// SIMATIC STEP 7 (V5.x) project PID_INS
// program: S7 Program(1)

SYMBOL_TABLE
"PID_L"	FB 136	FB 136	// Регулирования уровня в резервуаре активного ила
END_SYMBOL_TABLE

FUNCTION_BLOCK "PID_L"	// FB 136
AUTHOR : ETSystem
VERSION : 0.1
VAR_INPUT
  MAN_ON : BOOL ;
  P_SEL : BOOL ;
  I_SEL : BOOL ;
  D_SEL : BOOL ;
  SP_INT : REAL ;
  PV_IN : REAL ;
  MAN : REAL ;
  K_GAIN : REAL ;
  TI : TIME ;
  TD : TIME ;
  DEAD_BANDW : REAL ;
  LMN_HLM : REAL ;
  LMN_LLM : REAL ;
END_VAR
VAR_OUTPUT
  LMN : REAL ;
  PV : REAL ;
  ER : REAL ;
END_VAR
BEGIN
NETWORK
TITLE =
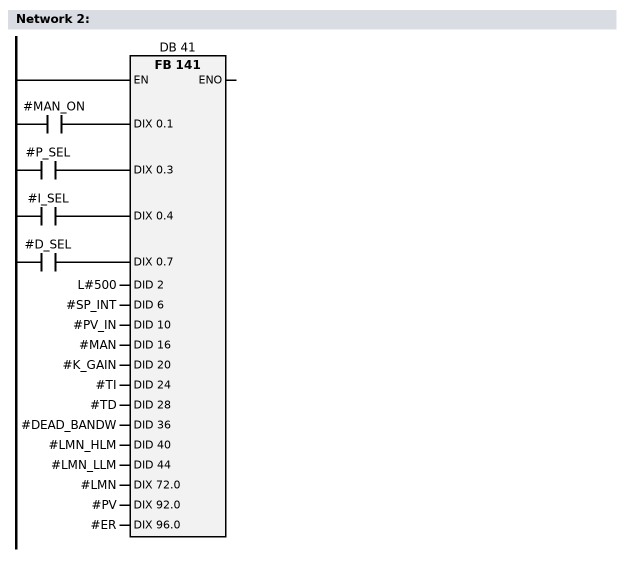
NETWORK
TITLE =
      A     #MAN_ON;
      =     L 0.1;
      BLD   103;
      A     #P_SEL;
      =     L 0.3;
      BLD   103;
      A     #I_SEL;
      =     L 0.4;
      BLD   103;
      A     #D_SEL;
      =     L 0.7;
      BLD   103;
      CALL  FB 141 , DB 41 (
           DIX 0.1                  := L 0.1,
           DIX 0.3                  := L 0.3,
           DIX 0.4                  := L 0.4,
           DIX 0.7                  := L 0.7,
           DID 2                    := L#500,
           DID 6                    := #SP_INT,
           DID 10                   := #PV_IN,
           DID 16                   := #MAN,
           DID 20                   := #K_GAIN,
           DID 24                   := #TI,
           DID 28                   := #TD,
           DID 36                   := #DEAD_BANDW,
           DID 40                   := #LMN_HLM,
           DID 44                   := #LMN_LLM,
           DIX 72.0                 := #LMN,
           DIX 92.0                 := #PV,
           DIX 96.0                 := #ER);
      NOP   0;
END_FUNCTION_BLOCK

ORGANIZATION_BLOCK OB 1
TITLE = "Main Program Sweep (Cycle)"
VERSION : 0.1
VAR_TEMP
  OB1_EV_CLASS : BYTE ;	//Bits 0-3 = 1 (Coming event), Bits 4-7 = 1 (Event class 1)
  OB1_SCAN_1 : BYTE ;	//1 (Cold restart scan 1 of OB 1), 3 (Scan 2-n of OB 1)
  OB1_PRIORITY : BYTE ;	//Priority of OB Execution
  OB1_OB_NUMBR : BYTE ;	//1 (Organization block 1, OB1)
  OB1_RESERVED_1 : BYTE ;	//Reserved for system
  OB1_RESERVED_2 : BYTE ;	//Reserved for system
  OB1_PREV_CYCLE : INT ;	//Cycle time of previous OB1 scan (milliseconds)
  OB1_MIN_CYCLE : INT ;	//Minimum cycle time of OB1 (milliseconds)
  OB1_MAX_CYCLE : INT ;	//Maximum cycle time of OB1 (milliseconds)
  OB1_DATE_TIME : DATE_AND_TIME ;	//Date and time OB1 started
END_VAR
BEGIN
// (block stored without names or comments; labels and parameter names are numbered)
END_ORGANIZATION_BLOCK
